FUNCTION_BLOCK FB_Ablauf
VAR_INPUT
	currentState: 	ST_SystemState;
END_VAR
VAR_OUTPUT
END_VAR
VAR
	iStep: 			INT := 000;
END_VAR

IF currentState.systemRUN THEN
	iStep := 010;
END_IF

CASE iStep OF
	
000: 				//INIT



END_CASE

END_FUNCTION_BLOCK

(* stored: Version 1.1.0.1
   POU FB_Ablauf: Id {1522559e-d157-41a8-a0be-2b09dc81f45b}, SpecialFunc None *)
